FUNCTION_BLOCK FB_FreqMeasure
// This function is the equivalent of FREQ_MEASURE from codesys's utility library
VAR_INPUT
	// Input signal
    IN: BOOL;
	// Number of periods to average the frequency over.
	// Must be between 1 and 100
    PERIODS: INT :=1;
	// Reset all parameters to 0
    RESET: BOOL;
END_VAR
VAR_OUTPUT
	// Frequency in HZ
    OUT: REAL;
	// FALSE until we've measured at least PERIODS periods, or if distance between two rising edges is > 3 * OUT
    VALID: BOOL;
END_VAR
VAR
	RisingEnableEdge: R_TRIG;
	FallingEnableEdge : F_TRIG;
    STARTED: BOOL;
    RISETIME: TIME;
	// Difference in time between current and last rising edge
    DIFF: DINT;
	// Array of time differences for each period
    TIMEDIFF: ARRAY[0..99] OF DINT;
	// How many periods we have counted so far
    COUNT: INT;
	// Current place in the array of time differences
    IDX: INT;
    I: INT;
	SUM: DINT;
	SYSTIMEMS : TIME;          
END_VAR


IF RESET THEN
    VALID := FALSE;
    COUNT := 0;
    IDX := 0;
    STARTED := FALSE;
    OUT := 0;
    RETURN;
END_IF

RisingEnableEdge(CLK := IN);
FallingEnableEdge(CLK := IN);

// We care only about whether we are the beginning or the end of the signal
IF RisingEnableEdge.Q OR FallingEnableEdge.Q THEN
	SYSTIMEMS := ULINT_TO_TIME(F_GetTaskTime() / TC2_Utilities.SYSTEMTIME_TICKSPERMSEC64);
    IF FallingEnableEdge.Q AND STARTED THEN
		DIFF := TIME_TO_DINT(SYSTIMEMS - RISETIME);
		// We assume time never goes backwards for real. Unfortunately, the API of this call does
		// not give us a way to express errors easily.
        IF Diff > 0 THEN
			// Emulate the weird behavior of CODESYS FREQ_MEASURE
			IF VALID AND Diff > 3000 * REAL_TO_DINT(OUT) THEN
				VALID := FALSE;
				COUNT := 0;
				IDX := 0;
				RETURN;
			END_IF
            TIMEDIFF[IDX] := DIFF;
            IDX := (IDX + 1) MOD PERIODS;
            COUNT := MIN(COUNT + 1, PERIODS);
			// Go valid once we have the minimum number of periods to average over.
            IF COUNT = PERIODS THEN
                SUM := 0;
				// Sum first, then convert to real, to minimize error.
                FOR I :=0 TO PERIODS-1 DO
                    SUM := SUM + TIMEDIFF[I];
                END_FOR
                OUT := 1000.0 * PERIODS / DINT_TO_REAL(SUM);
                VALID := TRUE;
            ELSE 
                VALID := FALSE;
            END_IF
        END_IF
		STARTED := FALSE;
		RETURN;
    END_IF
    STARTED := TRUE;
    RISETIME := SYSTIMEMS;
END_IF

END_FUNCTION_BLOCK

(* stored: Version 1.1.0.1, ProductVersion 3.1.4022.16
   POU FB_FreqMeasure: Id {3d6d3d65-e18a-4fc3-a773-f23be8247d43}, SpecialFunc None *)
